% RSLogix 500 project MIXING ROOM_BAK002.RSS, saved by version 11.00.00.00 %
PROJECT "UNTITLED"    % processor: MicroLogix 1200 %

PROGRAM FILES
  LAD 2   33 rungs

DATA FILES
  O0 OUTPUT  4 elements
  I1 INPUT  17 elements
  S2 STATUS  66 elements
  B3 BINARY  5 elements
  T4 TIMER  5 elements
  C5 COUNTER  1 elements
  R6 CONTROL  1 elements
  N7 INTEGER  60 elements
  F8 FLOAT  141 elements
  PD9   1 elements

LADDER 2
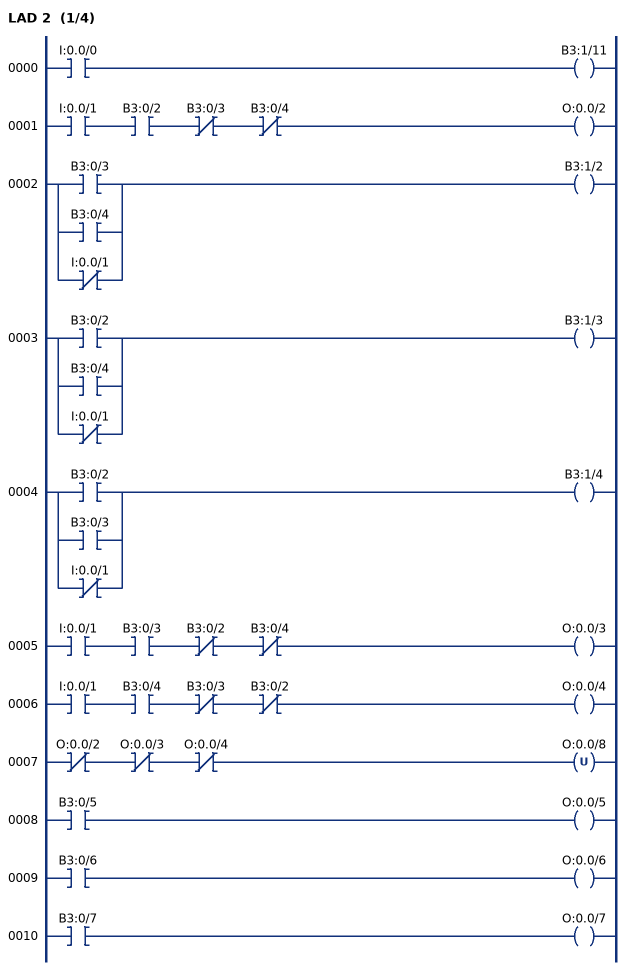
% Rung: 0 %
SOR XIC I:0.0/0 OTE B3:1/11 EOR
% Rung: 1 %
SOR XIC I:0.0/1 XIC B3:0/2 XIO B3:0/3 XIO B3:0/4 OTE O:0.0/2 EOR
% Rung: 2 %
SOR BST XIC B3:0/3 NXB BST XIC B3:0/4 NXB XIO I:0.0/1 BND BND OTE B3:1/2 EOR
% Rung: 3 %
SOR BST XIC B3:0/2 NXB BST XIC B3:0/4 NXB XIO I:0.0/1 BND BND OTE B3:1/3 EOR
% Rung: 4 %
SOR BST XIC B3:0/2 NXB BST XIC B3:0/3 NXB XIO I:0.0/1 BND BND OTE B3:1/4 EOR
% Rung: 5 %
SOR XIC I:0.0/1 XIC B3:0/3 XIO B3:0/2 XIO B3:0/4 OTE O:0.0/3 EOR
% Rung: 6 %
SOR XIC I:0.0/1 XIC B3:0/4 XIO B3:0/3 XIO B3:0/2 OTE O:0.0/4 EOR
% Rung: 7 %
SOR XIO O:0.0/2 XIO O:0.0/3 XIO O:0.0/4 OTU O:0.0/8 EOR
% Rung: 8 %
SOR XIC B3:0/5 OTE O:0.0/5 EOR
% Rung: 9 %
SOR XIC B3:0/6 OTE O:0.0/6 EOR
% Rung: 10 %
SOR XIC B3:0/7 OTE O:0.0/7 EOR

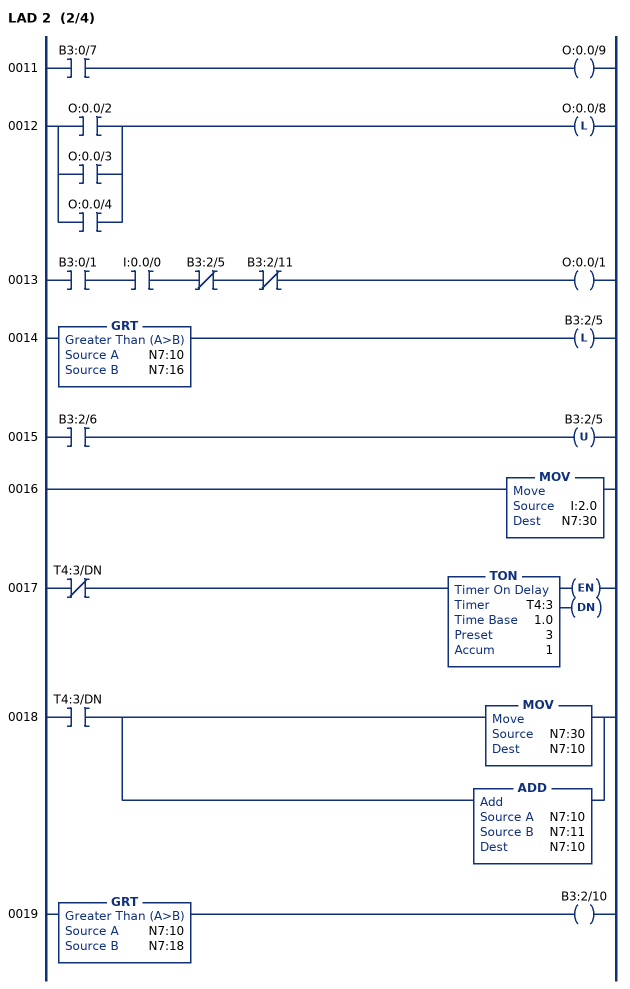
% Rung: 11 %
SOR XIC B3:0/7 OTE O:0.0/9 EOR
% Rung: 12 %
SOR BST XIC O:0.0/2 NXB BST XIC O:0.0/3 NXB XIC O:0.0/4 BND BND OTL O:0.0/8 EOR
% Rung: 13 %
SOR XIC B3:0/1 XIC I:0.0/0 XIO B3:2/5 XIO B3:2/11 OTE O:0.0/1 EOR
% Rung: 14 %
SOR GRT N7:10 N7:16 OTL B3:2/5 EOR
% Rung: 15 %
SOR XIC B3:2/6 OTU B3:2/5 EOR
% Rung: 16 %
SOR MOV I:2.0 N7:30 EOR
% Rung: 17 %
SOR XIO T4:3/DN TON T4:3 1.0 3 1 EOR
% Rung: 18 %
SOR XIC T4:3/DN BST MOV N7:30 N7:10 NXB ADD N7:10 N7:11 N7:10 BND EOR
% Rung: 19 %
SOR GRT N7:10 N7:18 OTE B3:2/10 EOR

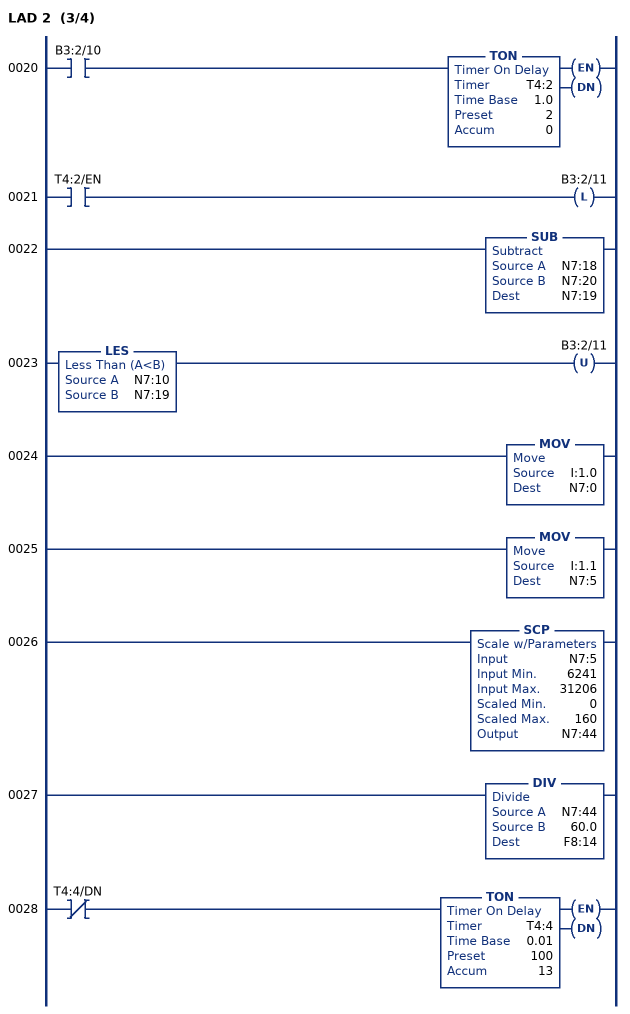
% Rung: 20 %
SOR XIC B3:2/10 TON T4:2 1.0 2 0 EOR
% Rung: 21 %
SOR XIC T4:2/EN OTL B3:2/11 EOR
% Rung: 22 %
SOR SUB N7:18 N7:20 N7:19 EOR
% Rung: 23 %
SOR LES N7:10 N7:19 OTU B3:2/11 EOR
% Rung: 24 %
SOR MOV I:1.0 N7:0 EOR
% Rung: 25 %
SOR MOV I:1.1 N7:5 EOR
% Rung: 26 %
SOR SCP N7:5 6241 31206 0 160 N7:44 EOR
% Rung: 27 %
SOR DIV N7:44 60.0 F8:14 EOR
% Rung: 28 %
SOR XIO T4:4/DN TON T4:4 0.01 100 13 EOR

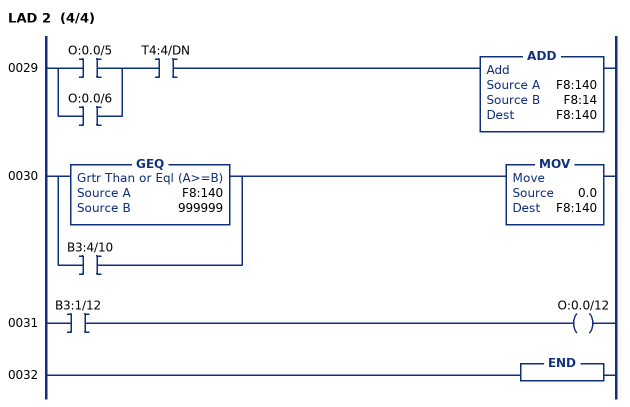
% Rung: 29 %
SOR BST XIC O:0.0/5 NXB XIC O:0.0/6 BND XIC T4:4/DN ADD F8:140 F8:14 F8:140 EOR
% Rung: 30 %
SOR BST GEQ F8:140 999999 NXB XIC B3:4/10 BND MOV 0.0 F8:140 EOR
% Rung: 31 %
SOR XIC B3:1/12 OTE O:0.0/12 EOR
% Rung: 32 %
SOR END EOR

DATA TABLE (non-zero values as saved)
DATA B3
% B3:0 % 0X0400 0X081C 0X0020 0X0000 0X0000
DATA T4
% .PRE .ACC %
% T4:1 % 15 0
% T4:2 % 2 0
% T4:3 % 3 1
% T4:4 % 100 13
DATA N7
% N7:0 % 11944 0 100 0 0 6248 0 100 0 0
% N7:10 % 66 0 1 1 0 0 275 0 160 155
% N7:20 % 5 0 0 0 0 0 0 0 0 0
% N7:30 % 77 0 0 0 0 0 0 0 0 0
% N7:50 % 0 0 0 0 0 0 0 0 0 18
